// TIA Portal V17 export
// export: Created 2024-08-29T18:23:49.1387045Z, ExportSetting WithDefaults, DisplayName Totally Integrated Automation Portal, DisplayVersion V17 Update 7, DisplayName TIA Portal Openness, DisplayVersion V17 Update 7, DisplayName TIA Portal Version Control Interface, DisplayVersion V17, DisplayName SINAMICS Startdrive Advanced, DisplayVersion V17 SP2, DisplayName SINAMICS Startdrive G110M, G120, G120C, G120D, G120P, G115D, DisplayVersion V17 SP2, DisplayName SINAMICS Startdrive G130, G150, S120, S150, SINAMICS MV, S210, DisplayVersion V17 SP2, DisplayName STEP 7 Professional, DisplayVersion V17 Update 7, DisplayName STEP 7 Safety, DisplayVersion V17 Update 6, DisplayName WinCC Advanced / Unified PC, DisplayVersion V17 Update 7
DATA_BLOCK "Receive_P2P_DB"   // DB28
// stored: AutoNumber true, DBAccessibleFromOPCUA true, DBAccessibleFromWebserver true, InstanceOfName Receive_P2P, OfSystemLibElement Receive_P2P, OfSystemLibVersion 1.4
"Receive_P2P"
   // VAR_INPUT
   //    PORT : PORT := 306;
   //    BUFFER : Variant;
   // END_VAR
   // VAR_OUTPUT
   //    NDR : Bool := FALSE;
   //    ERROR : Bool := FALSE;
   //    STATUS : Word := 16#7002;
   //    LENGTH : UInt := 0;
   // END_VAR
   // VAR
   //    OldPORT : PORT := 306;
   //    received_length : UInt := 16;
   //    y_ptp_status : SInt := 0;
   //    y_state : SInt := 0;
   //    y_seq_nr : Byte := 16#2E;
   //    safe_h1 : Byte := 16#00;
   //    safe_h2 : Byte := 16#00;
   //    safe_h3 : Byte := 16#00;
   //    safe_h4 : Byte := 16#00;
   //    isClassic : Bool := FALSE;
   //    record_nr : Int := 49;
   //    offset : UDInt := 0;
   //    RDREC { S7_SetPoint := 'True'} : RDREC;
   //    ReceiveBuffer : Array[0..1027] of Byte;
   //    i_addr : UDInt := 6;
   //    mySrcVAREF { ExternalAccessible := 'False'; ExternalVisible := 'False'; ExternalWritable := 'False'; S7_SetPoint := 'True'} : VAREF;
   //    myDstVAREF { ExternalVisible := 'False'; S7_SetPoint := 'True'} : VAREF;
   // END_VAR
BEGIN
   RDREC.REQ := FALSE;
   RDREC.ID := 306;
   RDREC.INDEX := 50;
   RDREC.MLEN := 1028;
   RDREC.VALID := TRUE;
   RDREC.BUSY := FALSE;
   RDREC.ERROR := FALSE;
   RDREC.STATUS := 16#0000_0000;
   RDREC.LEN := 20;
   ReceiveBuffer[0] := 16#2E;
   ReceiveBuffer[1] := 16#01;
   ReceiveBuffer[2] := 16#00;
   ReceiveBuffer[3] := 16#10;
   ReceiveBuffer[4] := 16#30;
   ReceiveBuffer[5] := 16#33;
   ReceiveBuffer[6] := 16#38;
   ReceiveBuffer[7] := 16#30;
   ReceiveBuffer[8] := 16#34;
   ReceiveBuffer[9] := 16#30;
   ReceiveBuffer[10] := 16#37;
   ReceiveBuffer[11] := 16#33;
   ReceiveBuffer[12] := 16#47;
   ReceiveBuffer[13] := 16#4F;
   ReceiveBuffer[14] := 16#32;
   ReceiveBuffer[15] := 16#33;
   ReceiveBuffer[16] := 16#35;
   ReceiveBuffer[17] := 16#34;
   ReceiveBuffer[18] := 16#38;
   ReceiveBuffer[19] := 16#0D;
   ReceiveBuffer[20] := 16#38;
   ReceiveBuffer[21] := 16#35;
   ReceiveBuffer[22] := 16#0D;
   ReceiveBuffer[23..1027] := 16#00;
   mySrcVAREF.RID := 16#0000_0000;
   mySrcVAREF.AREA := 16#00;
   mySrcVAREF.DB_NUMBER := 0;
   mySrcVAREF.OFFSET := 0;
   mySrcVAREF.LENGTH := 0;
   myDstVAREF.RID := 16#0201_0002;
   myDstVAREF.AREA := 16#8B;
   myDstVAREF.DB_NUMBER := 6;
   myDstVAREF.OFFSET := 2184;
   myDstVAREF.LENGTH := 255;
END_DATA_BLOCK
